(* PLC project SpindleLib, Delta Electronics, Inc. DIADesigner-AX DIADesigner-AX 1.3, author Piotr Gliszczyński *)
(* stored: creationDateTime 2022-11-02T13:12:47.6800751, version 3.5.15.30, modificationDateTime 2022-11-02T13:12:38.4366935, organization Induprogress *)
(* This Library allows to control spindles with simple FB. If you need to add another spindle option - just extend SpindleManager *)

{attribute 'qualified_only'}
{attribute 'strict'}
TYPE SpindleMaganerStatus_e : (INIT := 0, STANDBY, POWER_ON, WORKING_CW, WORKING_CCW, STOPPING, ERROR, DEFAULT := 9999);
END_TYPE

{attribute 'qualified_only'}
VAR_GLOBAL CONSTANT  (* Constants - {attribute 'conditionalshow'} {attribute 'conditionalshow' := 'SomeText'} {attribute 'hide'} *)
  DEFAULT_RAMP_TIME : REAL := 0.5;  (* default ramp time in seconds *)
  SP_DEFAULT_STATUS : SpindleMaganerStatus_e := SpindleMaganerStatus_e.DEFAULT;  (* default status of spindle state machine *)
  DEFAULT_MAX_VELOCITY : INT := 1500;  (* default max rotating speed of a spindle motor in RPM *)
END_VAR

INTERFACE ErrorInterface
METHOD errorReset : BOOL
END_METHOD
PROPERTY isError : BOOL
END_PROPERTY
END_INTERFACE

INTERFACE MotionInterface
METHOD setPowerOn
END_METHOD
METHOD runSpindle
  VAR_INPUT
    i_setVelocity : INT;
  END_VAR
END_METHOD
METHOD stopSpindle
END_METHOD
METHOD setPowerOff
END_METHOD
PROPERTY isPowerOn : BOOL
END_PROPERTY
PROPERTY isSpindleStopped : BOOL
END_PROPERTY
PROPERTY isSpindleTargetReached : BOOL
END_PROPERTY
END_INTERFACE

INTERFACE RampsInterface
METHOD writeRamps : BOOL
END_METHOD
METHOD rampsWasChanged : BOOL
END_METHOD
END_INTERFACE

(* * Class that enables to create objects - analog controlled spindles. Class extends general abstract implementation of spindles, with analog handling. * Class requires several additional signals from the drive - drive in error status, drive in power on status, drive stopped, drive target reached and actual veclity read from drive * Similarly, additional signals will be necesary to implement as outputs - drive reset, drive enable and obviously, drive analog signal. * * Class directly follows abstract class logic, if any override occurs - see description near override. Class implements Error and Motion interfaces. * Ramps interface is not necessary, since no ramps can be changed without communication. Ramps are set as constant in drive. * * Extend this block if any different behaviour is necessary *)
FUNCTION_BLOCK AnalogSpindle EXTENDS SpindleManager
  VAR_INPUT
    i_driveInError : BOOL;  (* feedback signals from drive *)
    i_drivePowerON : BOOL;
    i_driveStopped : BOOL;
    i_driveTargetReached : BOOL;
    i_driveActualVelocity : INT;
  END_VAR
  VAR_OUTPUT
    q_driveReset : BOOL;  (* signals sent to drive *)
    q_driveEnable : BOOL;  (* Power stage enable or servo ON *)
    q_driveAnalogCommand : INT;  (* analog rotating command. By default is sait to be signed, if unsigned command necessary extend and ovverride this class. *)
  END_VAR

            SUPER^( i_runCW := THIS^.i_runCW,
		i_runCCW := THIS^.i_runCCW,
		i_reset := THIS^.i_reset,
		i_targetVelocity := THIS^.i_targetVelocity,
		q_actualVelocity => THIS^.q_actualVelocity,
		q_error => THIS^.q_error,
		q_spindleStopped => THIS^.q_spindleStopped,
		q_spindleTargetReached => THIS^.q_spindleTargetReached);
          

(* * Analog spindle class method, handles error resets. IF called - outputs specific error reset output signal to the drive * When error is succesfully reset - returns TRUE. *)
METHOD errorReset : BOOL
                  THIS^.q_driveReset := isError;
IF NOT isError THEN
	errorReset := TRUE;
END_IF
                
END_METHOD

(* * Analog spindle implementation of motion interface - enables output which handlesc drive power stage control *)
METHOD setPowerOn
                  THIS^.q_driveEnable := TRUE;
                
END_METHOD

(* * Analog spindle implementation of motion interface method, handles running spindle. * Sets commadn to analog output and assumes signed analog output, if such implementation is not proper - override this method. *)
METHOD runSpindle
  VAR_INPUT
    i_setVelocity : INT;
  END_VAR
                  THIS^.q_driveAnalogCommand := i_setVelocity;
                
END_METHOD

(* * Analog spindle implementation of motion interface, handles stopping spindle by reseting (to 0) analog command *)
METHOD stopSpindle
                  THIS^.q_driveAnalogCommand := 0;
                
END_METHOD

(* * Analog spindle implementation of motion interface - disables output which handlesc drive power stage control *)
METHOD setPowerOff
                  THIS^.q_driveEnable := FALSE;
                
END_METHOD

(* * Overridden update method of spindle manager class. Override handles actual velocity output. *)
METHOD update
                  SUPER^.update();
THIS^.q_actualVelocity := THIS^.i_driveActualVelocity;
                
END_METHOD

(* * Analog spindle class method, handles reading error input from the drive - if it's true - drive is in error *)
PROPERTY isError : BOOL
GET
                    isError := THIS^.i_driveInError;
                  
END_GET
END_PROPERTY

(* * Analog spindle implementation of motion interface - checks input feedback from drive with powerON feedback *)
PROPERTY isPowerOn : BOOL
GET
                    isPowerOn := THIS^.i_drivePowerON;
                  
END_GET
END_PROPERTY

(* * Analog spindle implementation of motion interface - checks input feedback from drive with spindle stopped feedback *)
PROPERTY isSpindleStopped : BOOL
GET
                    isSpindleStopped := THIS^.i_driveStopped;
                  
END_GET
END_PROPERTY

(* * Analog spindle implementation of motion interface - checks input feedback from drive with target reacehd feedback *)
PROPERTY isSpindleTargetReached : BOOL
GET
                    isSpindleTargetReached := THIS^.i_driveTargetReached;
                  
END_GET
END_PROPERTY
END_FUNCTION_BLOCK

(* * Class that enables to create objects - modbus controlled spindles. Class extends general abstract implementation of spindles, with modbus communication handling. * Class requires several communication parameters to be read and mapped as inputs and outputs to the object. * * Class directly follows abstract class logic, if any override occurs - see description near override. Class implements Error, Motion and Ramps interfaces. * Ramps are imputs to the object by the user. Default implementation is necessary, since ramps cannot be 0. * * Any Delta Electronics VFD drive can be controlled with this block since modbus parameters are similar or the same in all models. Remember to set 00-20, 0-21 * and communication parameters in the drive * * Extend this block if any different behaviour is necessary *)
FUNCTION_BLOCK DeltaModbusSpindle EXTENDS SpindleManager
  VAR_INPUT
    i_warnErrorCode : UINT;  (* 2100h *)
    i_statusWord : UINT;  (* 2101h *)
    i_outputFrequency : INT;  (* 2102h *)
    i_accRamp : REAL := Constants.DEFAULT_RAMP_TIME;  (* input by user in s *)
    i_dccRamp : REAL := Constants.DEFAULT_RAMP_TIME;  (* input by user in s *)
  END_VAR
  VAR_OUTPUT
    q_controlWord : UINT;  (* 2000h *)
    q_frequencyCommand : INT;  (* 2001h *)
    q_driveReset : BOOL;  (* 2002.1h *)
    q_accRamp : UINT;  (* 01-12 = 010Ch *)
    q_dccRamp : UINT;  (* 01-13 = 010Dh *)
  END_VAR

            SUPER^( i_runCW := THIS^.i_runCW,
		i_runCCW := THIS^.i_runCCW,
		i_reset := THIS^.i_reset,
		i_targetVelocity := THIS^.i_targetVelocity,
		q_actualVelocity => THIS^.q_actualVelocity,
		q_error => THIS^.q_error,
		q_spindleStopped => THIS^.q_spindleStopped,
		q_spindleTargetReached => THIS^.q_spindleTargetReached);
          

(* * Modbus spindle method implementation of error interface - handles error reset, by enabling error reset output. * If reset succeeds returns TRUE *)
METHOD errorReset : BOOL
                  THIS^.q_driveReset := isError;
IF NOT isError THEN
	errorReset := TRUE;
END_IF
                
END_METHOD

(* * Modbus spindle ramps interface method implementation - handles sending ramps to drive. * * Since ramps in drive are scaled to 0.01s (1 = 0.01s) additional scaling was necessary and conversion from real to INT/UINT *)
METHOD writeRamps : BOOL
                  q_accRamp := TO_UINT(i_accRamp * 100);
q_dccRamp := TO_UINT(i_dccRamp * 100);

                
END_METHOD

(* * Modbus spindle ramps interface method implementation - handles checks if ramps set by user was changed, form what was sent to the drive * If input ramps are different, than output ramps - the user have changed ramp times and method returns TRUE * * Output ramps are integers with scaling 0.01s (1 = 0.01s), so additional scaling was necessary. *)
METHOD rampsWasChanged : BOOL
                  rampsWasChanged := (i_accRamp <> TO_REAL(q_accRamp)/100) OR (i_dccRamp <> TO_REAL(q_accRamp)/100);
                
END_METHOD

(* * Modbus spindle motion interface method implementation - starts the drive via specific controlwrod bits. *)
METHOD setPowerOn
                  THIS^.q_controlWord.0 := FALSE;
THIS^.q_controlWord.1 := TRUE;
                
END_METHOD

(* * Modbus spindle motion interface method implementation, handles running of the drive * - sending frequency command and selecting right rotation dricetion based on set vecloty *)
METHOD runSpindle
  VAR_INPUT
    i_setVelocity : INT;
  END_VAR
                  IF i_setVelocity >= 0 THEN
	THIS^.q_controlWord.4 := TRUE;
	THIS^.q_controlWord.5 := FALSE;
	THIS^.q_frequencyCommand := i_setVelocity;
ELSE
	THIS^.q_controlWord.4 := FALSE;
	THIS^.q_controlWord.5 := TRUE;
	THIS^.q_frequencyCommand := -i_setVelocity;
END_IF
                
END_METHOD

(* * Modbus spindle motion interface method implementation - stopps rotation of the spindle. Handled by 0 speed command. *)
METHOD stopSpindle
                  THIS^.q_frequencyCommand := 0;
                
END_METHOD

(* * Modbus spindle motion interface method implementation - stoppes the drive via specific controlwrod bits. *)
METHOD setPowerOff
                  THIS^.q_controlWord.0 := TRUE;
THIS^.q_controlWord.1 := FALSE;
                
END_METHOD

(* * Overridden update method of spindle manager class. Override handles actual velocity output. *)
METHOD update
                  SUPER^.update();
THIS^.q_actualVelocity := THIS^.i_outputFrequency;
                
END_METHOD

(* * Modbus spindle error interface property implementation - checks if drive reports any warn or error codes. If yes, then returns TRUE. *)
PROPERTY isError : BOOL
GET
                    IF THIS^.i_warnErrorCode <> 0 THEN
	isError := TRUE;
ELSE
	isError := FALSE;
END_IF
                  
END_GET
END_PROPERTY

(* * Modbus spindle motion interface property implementation - checks if any of the first two bits of control word is TRUE. * Returns true if yes - drive is in power ON state *)
PROPERTY isPowerOn : BOOL
GET
                    isPowerOn := (THIS^.i_statusWord.1 OR THIS^.i_statusWord.0);
                  
END_GET
END_PROPERTY

(* * Modbus spindle motion interface property implementation - checks if output frequency is 0 - if yesthe drive is stopped and returns TRUE *)
PROPERTY isSpindleStopped : BOOL
GET
                    isSpindleStopped := (THIS^.i_outputFrequency = 0);
                  
END_GET
END_PROPERTY

(* * Modbus spindle motion interface property implementation - handles checks of spindle target reached. * Checks if drive reports operating state and then checks if output frequency equals set frequency * Output frequency has 1.00Hz deadband implemented in checks *)
PROPERTY isSpindleTargetReached : BOOL
GET
                    isSpindleTargetReached := (THIS^.i_statusWord.0 AND THIS^.i_statusWord.1) AND 
(THIS^.i_outputFrequency <= THIS^.q_frequencyCommand + 100 OR THIS^.i_outputFrequency >= THIS^.q_frequencyCommand - 100);
                  
END_GET
END_PROPERTY
END_FUNCTION_BLOCK

(* * Class that enables to create EtherCAT controlled spindle drives. Class extends general implementation of abstract spindle manager class. * Class extends with etherCAT communication handling and thus needs several additional parameters maps. * * Class needs external inputs - ETCSlave (drive), status word, actual velocity - all of which are communication parameters. Ramp inputs are also necessary * Class outputs controlWord and target velocity all of which have to be mapped to communication parameters of the drive. * * Class directly follows abstract class logic, whith couple exceptions necessery for communication handling. If actual functionality is not enaugh - extend this class. *)
FUNCTION_BLOCK EthercatSpindle EXTENDS SpindleManager
  VAR_IN_OUT
    i_drive : ETCSlave;
  END_VAR
  VAR_INPUT
    i_statusWord : UINT;  (* 6041h - mapped from EtherCAT device *)
    i_actualVelocity : INT;  (* 606Ch - mapped from EtherCAT device *)
    i_accTime : REAL := Constants.DEFAULT_RAMP_TIME;  (* scaled in seconds *)
    i_dccTime : REAL := Constants.DEFAULT_RAMP_TIME;  (* scaled in seconds *)
  END_VAR
  VAR_OUTPUT
    q_controlWord : UINT;  (* 6040h - mapped to EtherCAT device *)
    q_targetVelocity : INT;  (* 60FFh - mapped to EtherCAT device *)
  END_VAR
  VAR
    OperationalDelay : TON;
    ReadAccRamp : ETC_CO_SdoRead := (wIndex := 16#3001, bySubindex := 16#D, pBuffer := ADR(accTimeRead), szSize := SIZEOF(accTimeRead));
    ReadDccRamp : ETC_CO_SdoRead := (wIndex := 16#3001, bySubindex := 16#E, pBuffer := ADR(dccTimeRead), szSize := SIZEOF(dccTimeRead));
    accTimeRead : INT;  (* ramps read from device *)
    dccTimeRead : INT;  (* ramps read from device *)
    WriteAccRamp : ETC_CO_SdoWrite := (wIndex := 16#604F, bySubindex := 16#0, pBuffer := ADR(accRamp), szSize := SIZEOF(accRamp));
    WriteDccRamp : ETC_CO_SdoWrite := (wIndex := 16#6050, bySubindex := 16#0, pBuffer := ADR(dccRamp), szSize := SIZEOF(dccRamp));
    accRamp : DINT;  (* ramps calculated by logic and sent to drive *)
    dccRamp : DINT;  (* ramps calculated by logic and sent to drive *)
  END_VAR

            IF OperationalDelay.Q THEN
	SUPER^( i_runCW := THIS^.i_runCW,
			i_runCCW := THIS^.i_runCCW,
			i_reset := THIS^.i_reset,
			i_targetVelocity := THIS^.i_targetVelocity,
			q_actualVelocity => THIS^.q_actualVelocity,
			q_error => THIS^.q_error,
			q_spindleStopped => THIS^.q_spindleStopped,
			q_spindleTargetReached => THIS^.q_spindleTargetReached);
END_IF;

//Delay of class logic to wait for communication start
OperationalDelay(IN:= (i_drive.wState = ETCStack.ETC_SLAVE_STATE.ETC_SLAVE_OPERATIONAL), PT:= T#1S);

//SDO FBs to read and send ramps via EtherCAT
//Default values are set, but can be changed if necessary
//Other values have to be set as seen below
//Unused values are unnecesary or used with FB.x operator
ReadAccRamp(
	usiCom:= 1, 
	uiDevice:= THIS^.i_drive.PhysSlaveAddr, 
	usiChannel:= 1,
	udiTimeOut := 100);

ReadDccRamp(
	usiCom:= 1, 
	uiDevice:= THIS^.i_drive.PhysSlaveAddr, 
	usiChannel:= 1,
	udiTimeOut := 100);
	
WriteAccRamp(
	usiCom:= 1, 
	uiDevice:= THIS^.i_drive.PhysSlaveAddr, 
	usiChannel:= 1, 
	udiTimeOut:= 100 );
	
WriteDccRamp(
	usiCom:= 1, 
	uiDevice:= THIS^.i_drive.PhysSlaveAddr, 
	usiChannel:= 1, 
	udiTimeOut:= 100 );
          

(* * Modbus spindle method implementation of error interface - handles error reset, by enabling bit 7 of controlword * If reset succeeds returns TRUE *)
METHOD errorReset : BOOL
                  THIS^.q_controlWord.7 := isError;
IF NOT isError THEN
	errorReset := TRUE;
END_IF 
                
END_METHOD

(* * EtherCAT spindle ramps interface method implementation - handles sending ramp times set by user to the drive * Ramps are set to the drive by SDO defined in FB. Both ramps are sent in one call of the method. * * Ramps sent to drive are scaled in ms and are DINTs. Input ramps have to be converted to DINT and scaled by 1000 *)
METHOD writeRamps : BOOL
                  THIS^.accRamp := TO_DINT(1000 * THIS^.i_accTime);
THIS^.dccRamp := TO_DINT(1000 * THIS^.i_dccTime);

THIS^.WriteAccRamp.xExecute := TRUE;

IF THIS^.WriteDccRamp.xDone OR THIS^.WriteDccRamp.xError OR THIS^.WriteAccRamp.xError THEN
	THIS^.WriteAccRamp.xExecute := FALSE;
	THIS^.WriteDccRamp.xExecute := FALSE;
END_IF

IF THIS^.WriteAccRamp.xDone THEN
	THIS^.WriteDccRamp.xExecute := TRUE;
END_IF

IF THIS^.WriteDccRamp.xExecute THEN
	writeRamps := TRUE;
END_IF
                
END_METHOD

(* * EtherCAT spindle ramps interface method implementation - handles checks if ramps set by user was changed, form what was read from the drive * If input ramps are different, than ramps currently in drive - the user have changed ramp times and method returns TRUE * * Ramps read form drive are integers with scaling 0.01s (1 = 0.01s), so additional scaling was necessary. * SDOs are read cyclicly in the method until both ramps were reads and boolean state of ramps is returned. *)
METHOD rampsWasChanged : BOOL
                  THIS^.ReadAccRamp.xExecute := TRUE;

IF THIS^.ReadAccRamp.xExecute AND THIS^.ReadAccRamp.xDone THEN
	IF TO_INT(THIS^.i_accTime*100) <> accTimeRead THEN
		rampsWasChanged := TRUE;
		THIS^.ReadAccRamp.xExecute := FALSE;
	ELSE
		THIS^.ReadDccRamp.xExecute := TRUE;
	END_IF
END_IF

IF THIS^.ReadDccRamp.xExecute AND THIS^.ReadDccRamp.xDone THEN
	IF TO_INT(THIS^.i_dccTime*100) <> dccTimeRead THEN
		rampsWasChanged := TRUE;
	ELSE
		rampsWasChanged := FALSE;
	END_IF
END_IF

IF THIS^.ReadDccRamp.xDone OR THIS^.ReadDccRamp.xError OR THIS^.ReadAccRamp.xError THEN
	THIS^.ReadAccRamp.xExecute := FALSE;
	THIS^.ReadDccRamp.xExecute := FALSE;
END_IF
	


                
END_METHOD

(* * EtherCAT spindle motion interface implementation methods - handling setting power stage ON , by seting of bit 0 of controlword *)
METHOD setPowerOn
                  THIS^.q_controlWord.0 := TRUE;
                
END_METHOD

(* * EtherCAT spindle motion interface implementation methods - handling running the spindle - setting target velocity and enabling operation (bits 4, 5, 6 of contorlword) *)
METHOD runSpindle
  VAR_INPUT
    i_setVelocity : INT;
  END_VAR
                  THIS^.q_targetVelocity := i_setVelocity;
THIS^.q_controlWord.4 := TRUE;
THIS^.q_controlWord.5 := TRUE;
THIS^.q_controlWord.6 := TRUE;
                
END_METHOD

(* * EtherCAT spindle motion interface implementation methods - handling stopping the spindle - setting target velocity to 0 * and disabling operation (bits 4, 5, 6 of contorlword) *)
METHOD stopSpindle
                  THIS^.q_targetVelocity := 0;
THIS^.q_controlWord.4 := FALSE;
THIS^.q_controlWord.5 := FALSE;
THIS^.q_controlWord.6 := FALSE;
                
END_METHOD

(* * EtherCAT spindle motion interface implementation methods - handling setting power stage OFF, by seting of bit 0 of controlword *)
METHOD setPowerOff
                  THIS^.q_controlWord.0 := FALSE;
                
END_METHOD

(* * Override of abstract method to handle output of actual veloctiy *)
METHOD update
                  SUPER^.update();
THIS^.q_actualVelocity := THIS^.i_actualVelocity;
                
END_METHOD

(* * Override of abstract method, so that the drive is initialized before standby status *)
METHOD standby
                  IF isInitialised THEN
	SUPER^.standby();
ELSE
	initDrive();
END_IF
                
END_METHOD

(* * EtherCAT spindle method, that extends standard motion interface. Via EtherCAT CiA402 drive by default is disabled (voltage is disabled, quick stop is disebled, etc) * The drive have to be disabled/enabled by user. This method is used to enale the drive - ie. after error reset to go back to default standby state. *)
METHOD initDrive
                  THIS^.q_controlWord.1 := TRUE;
THIS^.q_controlWord.2 := TRUE;
THIS^.q_controlWord.3 := TRUE;
                
END_METHOD

(* * EtherCAT spindle method, that extends standard motion interface. Via EtherCAT CiA402 drive by default is disabled (voltage is disabled, quick stop is disebled, etc) * The drive have to be disabled/enabled by user. This method is used to disabling the drive - ie. after error reset to go back to default standby state. *)
METHOD disableDrive
                  THIS^.q_controlWord.1 := FALSE;
THIS^.q_controlWord.2 := FALSE;
THIS^.q_controlWord.3 := FALSE;
                
END_METHOD

(* * Override of abstract method, so that the drive is disabled before initalization. Necessery to properly return from error state *)
METHOD initial : BOOL
                  disableDrive();
SUPER^.initial();
                
END_METHOD

(* * Modbus spindle error interface property implementation - checks if drive reports bit 3 or 7 in status word (error or warn). If yes, then returns TRUE. *)
PROPERTY isError : BOOL
GET
                    isError := THIS^.i_statusWord.3 OR THIS^.i_statusWord.7;
                  
END_GET
END_PROPERTY

(* * EtherCAT spindle motion interface property implementation - checks if drive reports servo ON bit (bit 1 of controlwrod). * If yes ther returns TRUE *)
PROPERTY isPowerOn : BOOL
GET
                    isPowerOn := THIS^.i_statusWord.1;
                  
END_GET
END_PROPERTY

(* * EtherCAT spindle motion interface property implementation - checks if drive reports that is stopped. * Property returns value TRUE if drive reports actual velocity = 9 *)
PROPERTY isSpindleStopped : BOOL
GET
                    isSpindleStopped := (THIS^.i_actualVelocity=0);
                  
END_GET
END_PROPERTY

(* * EtherCAT spindle motion interface property implementation - checks if drive reports that target is reached and actual velocity is different than 0 - * then returns true *)
PROPERTY isSpindleTargetReached : BOOL
GET
                    isSpindleTargetReached := (THIS^.i_actualVelocity<>0) AND THIS^.i_statusWord.10;
                  
END_GET
END_PROPERTY

(* * EtherCAT spindle motion interface property implementation - checks if drive reports proper status bits after initialisation * if all bits (0, 4, 5 of statusword) are present drive is initialized and method returns TRUE *)
PROPERTY isInitialised : BOOL
GET
                    isInitialised := THIS^.i_statusWord.0 AND THIS^.i_statusWord.4 AND THIS^.i_statusWord.5;
                  
END_GET
END_PROPERTY
END_FUNCTION_BLOCK

(* * Abstract class that represents general spindle. Spindle can be controlled via communication or analog signals - more precise implementation determines behaviour. * Generally, spindle usage in CNC machines is rather simple and in most applications it is only simple starting and stopping of the spindle. * This block represents this with spindle state machine, that could be - initialization, stadby, powered on, working - either CW or CCW, stopping or in error. * Furthermore couple of interfaces are implemented to include certain functionality - such as error handling or ramps handling. * * Block also requires certain inputs - run CW or CCW, reset and target speed of spindle in RPM and on the other hands return output with actual velocity, * error status, and spindle status (stopped or target reached). Additionally - actual velocity output does not have any implementation in abstract class, * since implementation might differ from spindle to spindle, yet the output is common to every spindle. Thus, developer have to implement it explicitly. * * Any other functionality (such as tool change positioning in more advanced spindles) or spindle behaviour can be achieved by extending this class. * * Override any class methods if implemented funcionality is too abstract or different behaviour is necessary. *)
FUNCTION_BLOCK SpindleManager IMPLEMENTS ErrorInterface, RampsInterface, MotionInterface
  VAR_INPUT
    i_runCW : BOOL;
    i_runCCW : BOOL;
    i_reset : BOOL;
    i_targetVelocity : UINT;  (* Target rotating speed in RPM *)
  END_VAR
  VAR_OUTPUT
    q_actualVelocity : INT;  (* Actual rotating speed in RPM *)
    q_error : BOOL;
    q_spindleStopped : BOOL;  (* Spindle is stopped and power stage is either ON or OFF *)
    q_spindleTargetReached : BOOL;  (* Target rotating speed has been reached *)
  END_VAR
  VAR
    status : SpindleMaganerStatus_e := 9999;
    nextStatus : SpindleMaganerStatus_e := SpindleMaganerStatus_e.INIT;
  END_VAR

            update(); //generally used for cyclic updating certain parameters - ie. ramps or status

CASE status OF
	SpindleMaganerStatus_e.INIT:
		initial(); //first cycles of the block or reset after error
	SpindleMaganerStatus_e.STANDBY:
		standby(); //drive has no error and is waiting ready for powering on
	SpindleMaganerStatus_e.POWER_ON:
		powerOn(); //drive is power and automatically goes into running state - either CW or CCW
	SpindleMaganerStatus_e.WORKING_CW:
		workingCW();
	SpindleMaganerStatus_e.WORKING_CCW:
		workingCCW();
	SpindleMaganerStatus_e.STOPPING:
		stopping();
	SpindleMaganerStatus_e.ERROR:
		error();
END_CASE
          

(* * Spindle manager abstract class method, handles updates of spindle manager. Updates status, ramps and outputs of this fb. * Additionally, if error occurs - proceeds to error state *)
METHOD update
                  //state machine status updates handling
THIS^.status := THIS^.nextStatus;

//error handling
IF NOT (status = SpindleMaganerStatus_e.INIT) THEN
	IF isError THEN
		nextStatus := SpindleMaganerStatus_e.ERROR;
	END_IF
END_IF;

//ramps updates if changed
IF rampsWasChanged() THEN
	writeRamps();
END_IF

//output handling
THIS^.q_error := isError;
THIS^.q_spindleStopped := isSpindleStopped;
THIS^.q_spindleTargetReached := isSpindleTargetReached;
                
END_METHOD

(* * Spindle manager abstact class method, handles initial state of spindle. If there are errors on the drives - the drive is reset and ramps are written. * Spindle then proceeds to standby state. If no error is present - only ramps are written and the proceeds to standby state *)
METHOD initial : BOOL
                  IF isError THEN
	IF errorReset() THEN
		IF writeRamps() THEN
			THIS^.nextStatus := SpindleMaganerStatus_e.STANDBY;
		END_IF
	END_IF
ELSE
	IF writeRamps() THEN
		THIS^.nextStatus := SpindleMaganerStatus_e.STANDBY;
	END_IF
END_IF
                
END_METHOD

METHOD errorReset : BOOL
                  
                
END_METHOD

METHOD writeRamps : BOOL
                  writeRamps := TRUE; //default implementation of the ramps for drives without ramps chaning or changing via drive parameters by service
                
END_METHOD

METHOD rampsWasChanged : BOOL
                  rampsWasChanged := FALSE; //default implementation of the ramps for drives without ramps chaning or changing via drive parameters by service
                
END_METHOD

(* * Spindle manager abstact class method, handles spindle in standby state. Generally, spindle is idle - wating for runnign command. Then proceeds to power on status *)
METHOD standby
                  IF THIS^.i_runCW OR THIS^.i_runCCW THEN
	THIS^.nextStatus := SpindleMaganerStatus_e.POWER_ON;
END_IF
                
END_METHOD

(* * Spindle manager abstract class method, handles spindle in power on status. If drive is not powered on - enables power. * Otherwise, proceeds to next states, which are either - working in any direction or stopping if run command is no longer present. *)
METHOD powerOn
                  IF NOT isPowerOn THEN
	setPowerOn();
ELSE
	IF THIS^.i_runCW THEN
		nextStatus := SpindleMaganerStatus_e.WORKING_CW;
	ELSIF THIS^.i_runCCW THEN
		nextStatus := SpindleMaganerStatus_e.WORKING_CCW;
	ELSE
		nextStatus := SpindleMaganerStatus_e.STOPPING;
	END_IF
END_IF
                
END_METHOD

METHOD setPowerOn : BOOL
                  
                
END_METHOD

(* * Spindle manager abstract class method, handles spindle in working in CW direction state. Enables the rotation with target velocity. * If direction command changes, directly switches the state. IF no command is present - proceeds to stopping state *)
METHOD workingCW
                  runSpindle(TO_INT(THIS^.i_targetVelocity));
IF NOT THIS^.i_runCW AND THIS^.i_runCCW THEN
	nextStatus := SpindleMaganerStatus_e.WORKING_CCW;
ELSIF NOT THIS^.i_runCW AND NOT THIS^.i_runCCW THEN
	nextStatus := SpindleMaganerStatus_e.STOPPING;
END_IF
                
END_METHOD

METHOD runSpindle : BOOL
  VAR_INPUT
    i_setPosition : INT;
  END_VAR
                  
                
END_METHOD

(* * Spindle manager abstract class method, handles spindle in working in CW direction state. Enables the rotation with target velocity. * Direction of rotating is handled by reversing target velocity command. * If direction command changes, directly switches the state. IF no command is present - proceeds to stopping state *)
METHOD workingCCW
                  runSpindle(-TO_INT(THIS^.i_targetVelocity));
IF NOT THIS^.i_runCCW AND THIS^.i_runCW THEN
	nextStatus := SpindleMaganerStatus_e.WORKING_CW;
ELSIF NOT THIS^.i_runCW AND NOT THIS^.i_runCCW THEN
	nextStatus := SpindleMaganerStatus_e.STOPPING;
END_IF
                
END_METHOD

(* * Spindla manager abstract class method, handles spindle in stopping state - disabels rotation of the spindle and when spindle is stopped, disables power stage * If spindle power stage is disabled - proceeds to standby state *)
METHOD stopping
                  IF NOT isSpindleStopped THEN
	stopSpindle();
ELSE
	setPowerOff();
END_IF

IF NOT isPowerOn THEN
	THIS^.nextStatus := SpindleMaganerStatus_e.STANDBY;
END_IF
                
END_METHOD

METHOD stopSpindle
                  
                
END_METHOD

METHOD setPowerOff
                  
                
END_METHOD

(* * Spindle Manager abstract class method, that handles spindle in error state. Disables stop and power on commands and waits for reset to change to initial state *)
METHOD error
                  IF THIS^.i_reset THEN
	THIS^.nextStatus:= SpindleMaganerStatus_e.INIT;
END_IF
stopSpindle();
setPowerOff();

                
END_METHOD

PROPERTY isError : BOOL
GET
                    
                  
END_GET
END_PROPERTY

PROPERTY isPowerOn : BOOL
GET
                    
                  
END_GET
END_PROPERTY

PROPERTY isSpindleStopped : BOOL
GET
                    
                  
END_GET
END_PROPERTY

PROPERTY isSpindleTargetReached : BOOL
GET
                    
                  
END_GET
END_PROPERTY
END_FUNCTION_BLOCK
